//----------------------------------------------------------------------------//
//            Copyright 2018 Rieckermann Engineering Operations               //
//                Automatically Generated File - Do Not Edit                  //
//----------------------------------------------------------------------------//
// Name:        ifbTI2                                                        //
// Description: Instances of TI2                                              //
//                                                                            //
// Line Mounted temperature Indicator.                                        //
//----------------------------------------------------------------------------//
// Revision history:                                                          //
// Rev By               Date        CC        Note                            //
// 2.0 David Paspa      08-Jan-2018 NA        Reboot for S7-1500.             //
// 0.3 Khairul Basar    17-Sep-2009 CC-09/016 USER_INPUT assigned to monitor. //
// 0.2 Khairul Basar    03-Sep-2009 CC-09/016 Initial value change-Ref.fbTI2. //
// 0.1 Khairul Basar    03-Aug-2009           Initial design.                 //
//----------------------------------------------------------------------------//
FUNCTION_BLOCK "ifbTI2"
TITLE = Instances of line mounted temperature indicator
{ S7_Optimized_Access := 'FALSE' }
AUTHOR : REO
NAME : ifbTI2
VERSION : 2.0

//----------------------------------------------------------------------------//
//                                                                            //
//----------------------------------------------------------------------------//
   VAR
@@TEMPLATE_BEGIN@@
      @@INSTANCE@@ : "fbTI2;   // @@DESCRIPTION@@
@@TEMPLATE_END@@
@@TEMPLATE_BEGIN@@
      @@INSTANCE@@_MODE : Struct
         PosEdge1 : Bool;
         PosEdge2 : Bool;
         REQ : Int;   // Request for Required Mode
      END_STRUCT;
@@TEMPLATE_END@@
   END_VAR

//----------------------------------------------------------------------------//
//                                                                            //
//----------------------------------------------------------------------------//
BEGIN
@@TEMPLATE_BEGIN@@
NETWORK
TITLE = @@INSTANCE@@ : @@DESCRIPTION@@
      A "alwaysHigh";
      = %L0.0;
      BLD 103;
      CALL "ifcTI2"
      (  IN_REQ_MODE                 := %L0.0 ,
         IN_MODE                     := "idb@@PARENTCLASS@@".@@PARENT@@_MODE.REQ ,
         OUT_MODE                    := #@@INSTANCE@@_MODE.REQ ,
         IO_MODE                     := "idbTI2".@@INSTANCE@@.MODE ,
         POS_EDGE1                   := #@@INSTANCE@@_MODE.PosEdge1 ,
         POS_EDGE2                   := #@@INSTANCE@@_MODE.PosEdge2
      );
      NOP 0;
NETWORK
TITLE = @@INSTANCE@@ : @@DESCRIPTION@@
      CALL #@@INSTANCE@@
      (  MODE                        := #@@INSTANCE@@.MODE ,
         RAW_INPUT                   := "P_TI-@@NUMINSTANCE@@":P ,
         USER_INPUT                  := #@@INSTANCE@@.USER_INPUT ,
         UPPER_RANGE                 := #@@INSTANCE@@.UPPER_RANGE ,
         LOWER_RANGE                 := #@@INSTANCE@@.LOWER_RANGE ,
         POLARITY                    := #@@INSTANCE@@.POLARITY ,
         LIMIT_HH                    := #@@INSTANCE@@.LIMIT_HH ,
         LIMIT_H                     := #@@INSTANCE@@.LIMIT_H ,
         LIMIT_L                     := #@@INSTANCE@@.LIMIT_L ,
         LIMIT_LL                    := #@@INSTANCE@@.LIMIT_LL ,
         ENABLE_HH                   := #@@INSTANCE@@.ENABLE_HH ,
         ENABLE_H                    := #@@INSTANCE@@.ENABLE_H ,
         ENABLE_L                    := #@@INSTANCE@@.ENABLE_L ,
         ENABLE_LL                   := #@@INSTANCE@@.ENABLE_LL ,
         MEASURE                     := #@@INSTANCE@@.MEASURE ,
         DATA_QUALITY                := #@@INSTANCE@@.DATA_QUALITY ,
         ALARM_HH                    := #@@INSTANCE@@.ALARM_HH ,
         ALARM_H                     := #@@INSTANCE@@.ALARM_H ,
         ALARM_L                     := #@@INSTANCE@@.ALARM_L ,
         ALARM_LL                    := #@@INSTANCE@@.ALARM_LL ,
         RANGE_ERROR                 := #@@INSTANCE@@.RANGE_ERROR ,
         BROKEN_WIRE                 := #@@INSTANCE@@.BROKEN_WIRE
      );
      NOP 0;
@@TEMPLATE_END@@
END_FUNCTION_BLOCK
